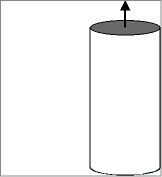
VISUALIZATION VISU_Tube_Top_13  // 162x177
VAR_IN_OUT
	azi : LREAL;
END_VAR
    Ellipse (90,160 70x15)
        p2858320360: azi
    Polygon (90,27) (160,27) (160,167) (154,171) (148,172) (141,174) (132,174) (121,174) (112,174) (104,173) (96,171) (90,167)
        p2858320360: azi
    Ellipse (90,20 70x15)
        p2858320360: azi
    Polygon (120,10) (125,0) (130,10)
        p2858320360: azi
    Polyline (125,27) (125,10)
        p2858320360: azi
    Polyline (160,168) (160,27)
        p2858320360: azi
    Polyline (90,168) (90,27)
        p2858320360: azi
END_VISUALIZATION

(* stored: Version 1.1.0.1, ProductVersion 3.1.4018.5
   Visu VISU_Tube_Top_13: Id {d5548d6f-001e-49c2-a000-8b64598e7ab4} *)
